// TIA Portal project "Assembler-Analog" (V15.1)

(* hardware
DEVICE "S7-1200 station_1"  S7-1200 Station
   slot 0: "Rack_0"  S7-1200 Rack  Rack  V1.0
   slot 1: "PLC_1"  CPU 1211C DC/DC/DC  6ES7 211-1AE40-0XB0  V4.2
DEVICE "HMI_1"  KTP900 Basic PN
   slot 0: "HMI_1"  KTP900 Basic PN  6AV2 123-2JB03-0AX0  15.1.0.0
   slot 1: "HMI_RT_1"  KTP900 Basic PN  6AV2 123-2JB03-0AX0  15.1.0.0
   slot 5: "HMI_1.IE_CP_1"  PROFINET Interface  15.0.1.0
      slot 1: "PROFINET Interface_1"  PROFINET Interface
         slot 1: "Port_1"  Port
*)

// ===== PLC "PLC_1"  CPU 1211C DC/DC/DC =====

VAR_GLOBAL   // PLC tag table "Default tag table"
   "Clock_Byte" AT %MB0 : Byte;
   "Clock_10Hz" AT %M0.0 : Bool;
   "Clock_5Hz" AT %M0.1 : Bool;
   "Clock_2.5Hz" AT %M0.2 : Bool;
   "Clock_2Hz" AT %M0.3 : Bool;
   "Clock_1.25Hz" AT %M0.4 : Bool;
   "Clock_1Hz" AT %M0.5 : Bool;
   "Clock_0.625Hz" AT %M0.6 : Bool;
   "Clock_0.5Hz" AT %M0.7 : Bool;
END_VAR

VAR_GLOBAL   // PLC tag table "IO_tags"
   "item_detected" AT %I0.0 : Bool;
   "lid_at_place" AT %I0.1 : Bool;
   "base_at_place" AT %I0.2 : Bool;
   "part_leaving" AT %I0.3 : Bool;
   "start" AT %I0.4 : Bool;
   "reset" AT %I0.5 : Bool;
   "stop" AT %I0.6 : Bool;
   "esd" AT %I0.7 : Bool;
   "auto" AT %I1.0 : Bool;
   "running" AT %I1.1 : Bool;
   "lids_conveyor_1" AT %Q0.0 : Bool;
   "stop_blade_1" AT %Q0.1 : Bool;
   "lids_conveyor_2" AT %Q0.2 : Bool;
   "base_conveyor_1" AT %Q0.3 : Bool;
   "stop_blade_2" AT %Q0.4 : Bool;
   "base_conveyor_2" AT %Q0.5 : Bool;
   "grab" AT %Q0.6 : Bool;
   "start_light" AT %Q0.7 : Bool;
   "reset_light" AT %Q1.0 : Bool;
   "stop_light" AT %Q1.1 : Bool;
   "x" AT %ID30 : Real;
   "z" AT %ID34 : Real;
   "set_x" AT %QD30 : Real;
   "set_z" AT %QD34 : Real;
   "counter" AT %QD38 : DInt;
END_VAR

DATA_BLOCK "Auxiliare"   // DB1
{ S7_Optimized_Access := 'TRUE' }
VERSION : 0.1
   VAR
      aux_1 : Bool;
      aux_2 : Bool;
      aux_3 : Bool;
      aux_4 : Bool;
      aux_5 : Bool;
      btn_reset_counter : Bool;
   END_VAR
BEGIN
END_DATA_BLOCK

DATA_BLOCK "Alarme"   // DB2
{ S7_Optimized_Access := 'TRUE' }
VERSION : 0.1
   VAR
      gather : Word;
      "array" : Array[0..15] of Bool;
   END_VAR
BEGIN
END_DATA_BLOCK

// folder: System blocks/Program resources

DATA_BLOCK "timer_reset_counter"   // DB3
{ S7_Optimized_Access := 'TRUE' }
AUTHOR : Simatic
FAMILY : IEC
NAME : IEC_TMR
VERSION : 1.0
// stored: InstanceOfName IEC_TIMER
"IEC_TIMER"
BEGIN
END_DATA_BLOCK

// folder: (top level)

FUNCTION "Analog_Assembler" : Void   // FC1, LAD
{ S7_Optimized_Access := 'TRUE' }
VERSION : 0.1
   VAR_TEMP   // added for the SCL form of the ladder/FBD networks
      _w1 : Bool;
      _w2 : Bool;
   END_VAR
BEGIN

REGION Network 1
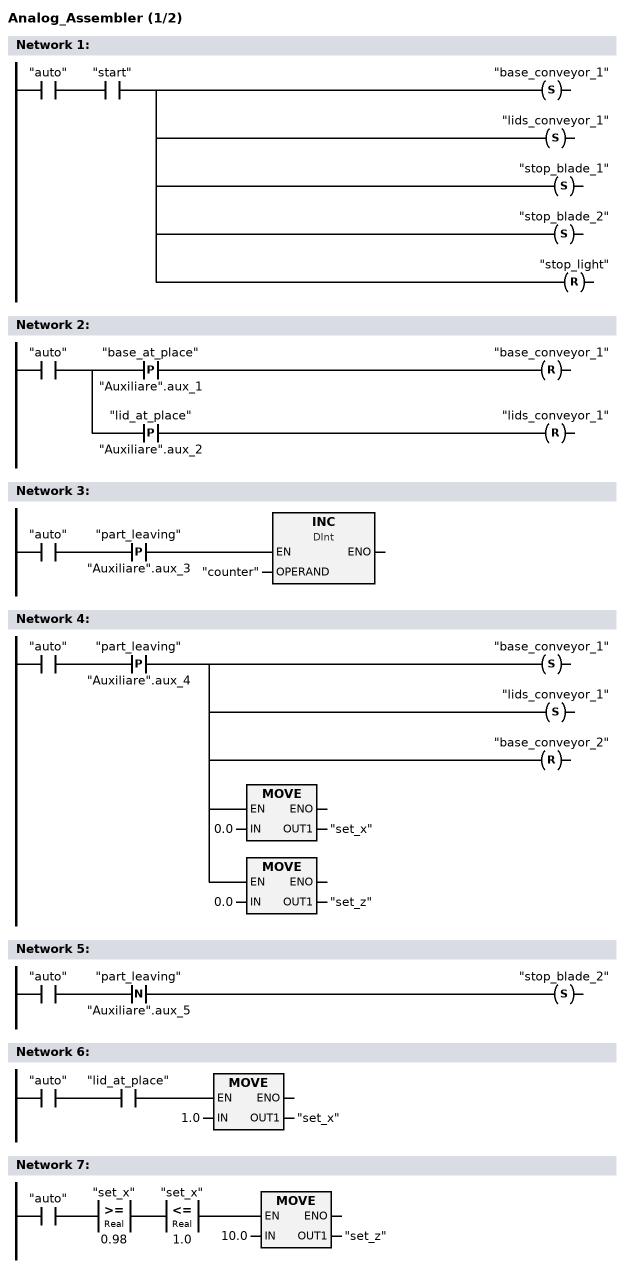
   RUNG wire#powerrail
      Contact( "auto" )
      Contact( "start" )
      wire#w1
      S_Coil( "base_conveyor_1" )
   END_RUNG
   RUNG wire#w1
      S_Coil( "lids_conveyor_1" )
   END_RUNG
   RUNG wire#w1
      S_Coil( "stop_blade_1" )
   END_RUNG
   RUNG wire#w1
      S_Coil( "stop_blade_2" )
   END_RUNG
   RUNG wire#w1
      R_Coil( "stop_light" )
   END_RUNG
   // the same network as SCL:
   IF "auto" AND "start" THEN
       "base_conveyor_1" := TRUE;
       "lids_conveyor_1" := TRUE;
       "stop_blade_1" := TRUE;
       "stop_blade_2" := TRUE;
       "stop_light" := FALSE;
   END_IF;
END_REGION

REGION Network 2
   RUNG wire#powerrail
      Contact( "auto" )
      wire#w1
      P_Contact(operand := "base_at_place", bit := "Auxiliare".aux_1)
      R_Coil( "base_conveyor_1" )
   END_RUNG
   RUNG wire#w1
      P_Contact(operand := "lid_at_place", bit := "Auxiliare".aux_2)
      R_Coil( "lids_conveyor_1" )
   END_RUNG
   // the same network as SCL:
   #_w1 := "auto" AND "base_at_place" AND NOT "Auxiliare".aux_1;   // rising edge of "base_at_place"
   "Auxiliare".aux_1 := "base_at_place";
   IF #_w1 THEN "base_conveyor_1" := FALSE; END_IF;
   #_w2 := "auto" AND "lid_at_place" AND NOT "Auxiliare".aux_2;   // rising edge of "lid_at_place"
   "Auxiliare".aux_2 := "lid_at_place";
   IF #_w2 THEN "lids_conveyor_1" := FALSE; END_IF;
END_REGION

REGION Network 3
   RUNG wire#powerrail
      Contact( "auto" )
      P_Contact(operand := "part_leaving", bit := "Auxiliare".aux_3)
      { S7_Templates := "DestType := DInt" } Inc( "counter" )
   END_RUNG
   // the same network as SCL:
   #_w1 := "auto" AND "part_leaving" AND NOT "Auxiliare".aux_3;   // rising edge of "part_leaving"
   "Auxiliare".aux_3 := "part_leaving";
   IF #_w1 THEN "counter" := "counter" + 1; END_IF;
END_REGION

REGION Network 4
   RUNG wire#powerrail
      Contact( "auto" )
      P_Contact(operand := "part_leaving", bit := "Auxiliare".aux_4)
      wire#w1
      S_Coil( "base_conveyor_1" )
   END_RUNG
   RUNG wire#w1
      S_Coil( "lids_conveyor_1" )
   END_RUNG
   RUNG wire#w1
      R_Coil( "base_conveyor_2" )
   END_RUNG
   RUNG wire#w1
      Move(in := 0.0, out1 => "set_x")
   END_RUNG
   RUNG wire#w1
      Move(in := 0.0, out1 => "set_z")
   END_RUNG
   // the same network as SCL:
   #_w1 := "auto" AND "part_leaving" AND NOT "Auxiliare".aux_4;   // rising edge of "part_leaving"
   "Auxiliare".aux_4 := "part_leaving";
   IF #_w1 THEN
       "base_conveyor_1" := TRUE;
       "lids_conveyor_1" := TRUE;
       "base_conveyor_2" := FALSE;
       "set_x" := 0.0;
       "set_z" := 0.0;
   END_IF;
END_REGION

REGION Network 5
   RUNG wire#powerrail
      Contact( "auto" )
      N_Contact(operand := "part_leaving", bit := "Auxiliare".aux_5)
      S_Coil( "stop_blade_2" )
   END_RUNG
   // the same network as SCL:
   #_w1 := "auto" AND NOT "part_leaving" AND "Auxiliare".aux_5;   // falling edge of "part_leaving"
   "Auxiliare".aux_5 := "part_leaving";
   IF #_w1 THEN "stop_blade_2" := TRUE; END_IF;
END_REGION

REGION Network 6
   RUNG wire#powerrail
      Contact( "auto" )
      Contact( "lid_at_place" )
      Move(in := 1.0, out1 => "set_x")
   END_RUNG
   // the same network as SCL:
   IF "auto" AND "lid_at_place" THEN "set_x" := 1.0; END_IF;
END_REGION

REGION Network 7
   RUNG wire#powerrail
      Contact( "auto" )
      { S7_Templates := "SrcType := Real" } GE_Contact(in1 := "set_x", in2 := 0.98)
      { S7_Templates := "SrcType := Real" } LE_Contact(in1 := "set_x", in2 := 1.0)
      Move(in := 10.0, out1 => "set_z")
   END_RUNG
   // the same network as SCL:
   IF "auto" AND ("set_x" >= 0.98) AND ("set_x" <= 1.0) THEN "set_z" := 10.0; END_IF;
END_REGION

REGION Network 8
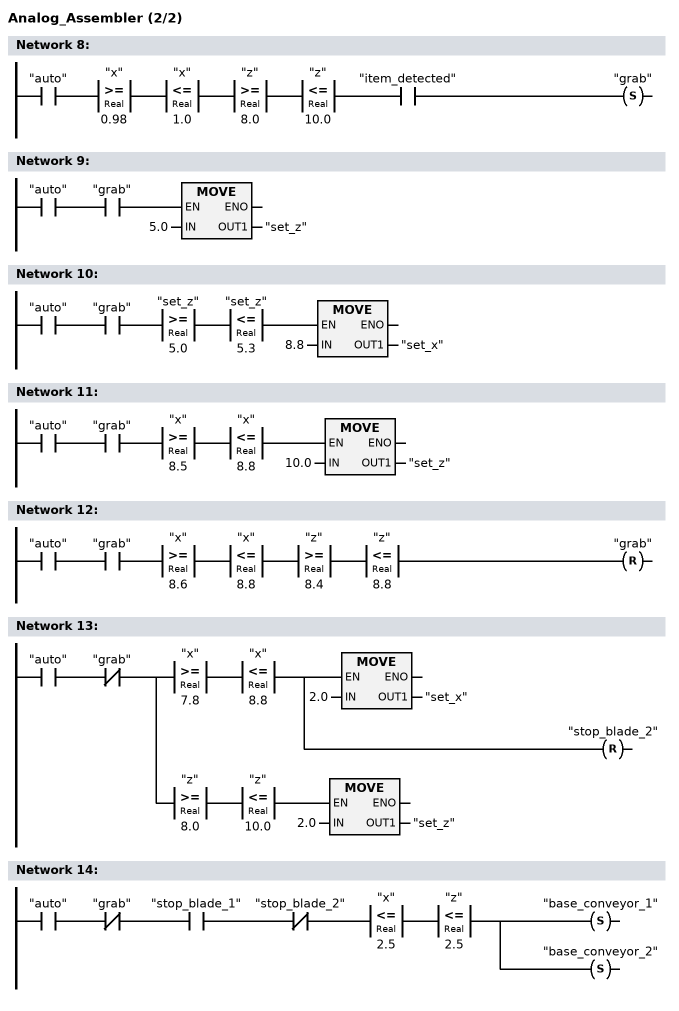
   RUNG wire#powerrail
      Contact( "auto" )
      { S7_Templates := "SrcType := Real" } GE_Contact(in1 := "x", in2 := 0.98)
      { S7_Templates := "SrcType := Real" } LE_Contact(in1 := "x", in2 := 1.0)
      { S7_Templates := "SrcType := Real" } GE_Contact(in1 := "z", in2 := 8.0)
      { S7_Templates := "SrcType := Real" } LE_Contact(in1 := "z", in2 := 10.0)
      Contact( "item_detected" )
      S_Coil( "grab" )
   END_RUNG
   // the same network as SCL:
   IF "auto" AND ("x" >= 0.98) AND ("x" <= 1.0) AND ("z" >= 8.0) AND ("z" <= 10.0) AND "item_detected" THEN
       "grab" := TRUE;
   END_IF;
END_REGION

REGION Network 9
   RUNG wire#powerrail
      Contact( "auto" )
      Contact( "grab" )
      Move(in := 5.0, out1 => "set_z")
   END_RUNG
   // the same network as SCL:
   IF "auto" AND "grab" THEN "set_z" := 5.0; END_IF;
END_REGION

REGION Network 10
   RUNG wire#powerrail
      Contact( "auto" )
      Contact( "grab" )
      { S7_Templates := "SrcType := Real" } GE_Contact(in1 := "set_z", in2 := 5.0)
      { S7_Templates := "SrcType := Real" } LE_Contact(in1 := "set_z", in2 := 5.3)
      Move(in := 8.8, out1 => "set_x")
   END_RUNG
   // the same network as SCL:
   IF "auto" AND "grab" AND ("set_z" >= 5.0) AND ("set_z" <= 5.3) THEN "set_x" := 8.8; END_IF;
END_REGION

REGION Network 11
   RUNG wire#powerrail
      Contact( "auto" )
      Contact( "grab" )
      { S7_Templates := "SrcType := Real" } GE_Contact(in1 := "x", in2 := 8.5)
      { S7_Templates := "SrcType := Real" } LE_Contact(in1 := "x", in2 := 8.8)
      Move(in := 10.0, out1 => "set_z")
   END_RUNG
   // the same network as SCL:
   IF "auto" AND "grab" AND ("x" >= 8.5) AND ("x" <= 8.8) THEN "set_z" := 10.0; END_IF;
END_REGION

REGION Network 12
   RUNG wire#powerrail
      Contact( "auto" )
      Contact( "grab" )
      { S7_Templates := "SrcType := Real" } GE_Contact(in1 := "x", in2 := 8.6)
      { S7_Templates := "SrcType := Real" } LE_Contact(in1 := "x", in2 := 8.8)
      { S7_Templates := "SrcType := Real" } GE_Contact(in1 := "z", in2 := 8.4)
      { S7_Templates := "SrcType := Real" } LE_Contact(in1 := "z", in2 := 8.8)
      R_Coil( "grab" )
   END_RUNG
   // the same network as SCL:
   IF "auto" AND "grab" AND ("x" >= 8.6) AND ("x" <= 8.8) AND ("z" >= 8.4) AND ("z" <= 8.8) THEN
       "grab" := FALSE;
   END_IF;
END_REGION

REGION Network 13
   RUNG wire#powerrail
      Contact( "auto" )
      I_Contact( "grab" )
      wire#w1
      { S7_Templates := "SrcType := Real" } GE_Contact(in1 := "x", in2 := 7.8)
      { S7_Templates := "SrcType := Real" } LE_Contact(in1 := "x", in2 := 8.8)
      wire#w2
      Move(in := 2.0, out1 => "set_x")
   END_RUNG
   RUNG wire#w2
      R_Coil( "stop_blade_2" )
   END_RUNG
   RUNG wire#w1
      { S7_Templates := "SrcType := Real" } GE_Contact(in1 := "z", in2 := 8.0)
      { S7_Templates := "SrcType := Real" } LE_Contact(in1 := "z", in2 := 10.0)
      Move(in := 2.0, out1 => "set_z")
   END_RUNG
   // the same network as SCL:
   #_w1 := "auto" AND NOT "grab";
   IF #_w1 AND ("x" >= 7.8) AND ("x" <= 8.8) THEN
       "set_x" := 2.0;
       "stop_blade_2" := FALSE;
   END_IF;
   IF #_w1 AND ("z" >= 8.0) AND ("z" <= 10.0) THEN "set_z" := 2.0; END_IF;
END_REGION

REGION Network 14
   RUNG wire#powerrail
      Contact( "auto" )
      I_Contact( "grab" )
      Contact( "stop_blade_1" )
      I_Contact( "stop_blade_2" )
      { S7_Templates := "SrcType := Real" } LE_Contact(in1 := "x", in2 := 2.5)
      { S7_Templates := "SrcType := Real" } LE_Contact(in1 := "z", in2 := 2.5)
      wire#w1
      S_Coil( "base_conveyor_1" )
   END_RUNG
   RUNG wire#w1
      S_Coil( "base_conveyor_2" )
   END_RUNG
   // the same network as SCL:
   IF "auto" AND NOT "grab" AND "stop_blade_1" AND NOT "stop_blade_2" AND ("x" <= 2.5) AND ("z" <= 2.5) THEN
       "base_conveyor_1" := TRUE;
       "base_conveyor_2" := TRUE;
   END_IF;
END_REGION
END_FUNCTION

FUNCTION "MHJ-PLC-Lab-Function-S71200" : Void   // FC9000, SCL
{ S7_Optimized_Access := 'TRUE' }
VERSION : 0.1
   VAR_TEMP
      rdTimeReturn : Int;
      outputTime : DTL;
      SyncVal : Byte;
      forVal : Int;
      forVal_2 : Int;
      Value : Byte;
   END_VAR
   VAR CONSTANT
      CompVal : Byte := 16#34;
      Value_01 : Byte := 16#11;
      Value_01_DW : DWord := 16#A165_D992;
      Value_02_DW : DWord := 16#58BE_4401;
   END_VAR
BEGIN

   #Value:=PEEK(area := 16#82,
        dbNumber := 0,
        byteOffset := 511);
   #Value := #Value + 1;

   POKE(area := 16#82,
        dbNumber := 0,
        byteOffset := 511,
        value := #Value);

   POKE(area:=16#81,
        dbNumber:=0,
        byteOffset:=1016,
        value:=#Value_01_DW);
   POKE(area := 16#81,
        dbNumber := 0,
        byteOffset := 1020,
        value := #Value_02_DW);

   POKE(area := 16#81,
        dbNumber := 0,
        byteOffset := 511,
        value := B#16#00);

   FOR #forVal := 0 TO 120 DO
       FOR #forVal_2:=0 TO 10 DO
           #rdTimeReturn:=RD_SYS_T(#outputTime);
           #rdTimeReturn := WR_SYS_T(#outputTime);
           #rdTimeReturn := RD_SYS_T(#outputTime);
           #rdTimeReturn := WR_SYS_T(#outputTime);
       END_FOR;
       #SyncVal:= PEEK(area := 16#81,
                      dbNumber := 0,
                      byteOffset := 511);
       IF #SyncVal = #CompVal THEN
          GOTO M_1;
       END_IF;
   END_FOR;
   RETURN;

   M_1:
   POKE(area := 16#81,
        dbNumber := 0,
        byteOffset := 511,
        value := B#16#0);
END_FUNCTION

ORGANIZATION_BLOCK "Main"   // OB1, LAD, ProgramCycle
TITLE = "Main Program Sweep (Cycle)"
{ S7_Optimized_Access := 'TRUE' }
VERSION : 0.1
   VAR_INPUT
      Initial_Call : Bool;   // Initial call of this OB
      Remanence : Bool;   // =True, if remanent data are available
   END_VAR
BEGIN

REGION Network 1: fct de conectare la factory io
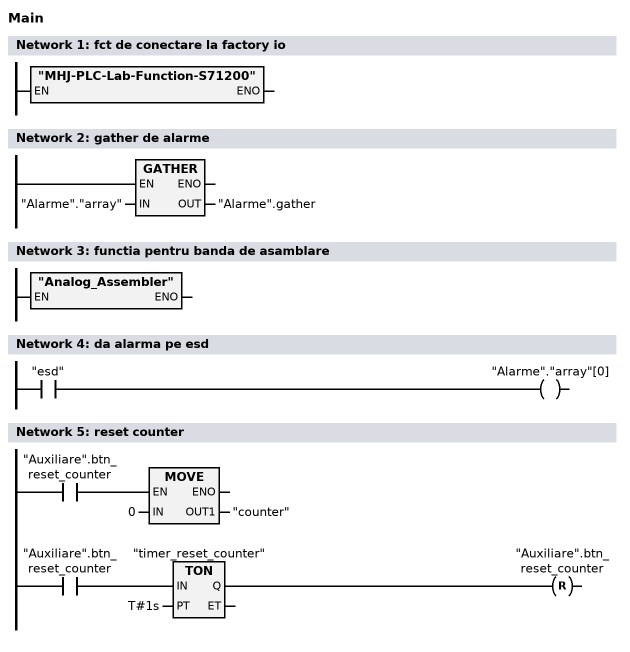
   RUNG wire#powerrail
      "MHJ-PLC-Lab-Function-S71200"()
   END_RUNG
   // the same network as SCL:
   "MHJ-PLC-Lab-Function-S71200"();
END_REGION

REGION Network 2: gather de alarme
   GATHER(IN := "Alarme"."array", OUT => "Alarme".gather);
END_REGION

REGION Network 3: functia pentru banda de asamblare
   RUNG wire#powerrail
      "Analog_Assembler"()
   END_RUNG
   // the same network as SCL:
   "Analog_Assembler"();
END_REGION

REGION Network 4: da alarma pe esd
   RUNG wire#powerrail
      Contact( "esd" )
      Coil( "Alarme"."array"[0] )
   END_RUNG
   // the same network as SCL:
   "Alarme"."array"[0] := "esd";
END_REGION

REGION Network 5: reset counter
   IF "Auxiliare".btn_reset_counter THEN "counter" := 0; END_IF;
   "timer_reset_counter".TON(IN := "Auxiliare".btn_reset_counter, PT := T#1s);
   IF "timer_reset_counter".Q THEN "Auxiliare".btn_reset_counter := FALSE; END_IF;
END_REGION
END_ORGANIZATION_BLOCK

(* ===== HMI "HMI_RT_1" =====
system functions are stored by id; their names below are inferred from use
connection "HMI_Connection_1": ETHERNET, SMART_S7_1200_OMS

HMI tags "Default tag table"
   "counter" : DInt = PLC counter AT %QD38, 1 s
   "Auxiliare_btn_reset_counter" : Bool = PLC Auxiliare.btn_reset_counter, 1 s
   "Alarme_gather" : Word = PLC Alarme.gather, 1 s

discrete alarms
   1: 'ESD', class Errors, trigger "Alarme_gather" bit 0

Template "Template_1" 800x480
   Button "Exit" at 722,440 size 55x39; TextOff 'Exit'; PictureOff "ExitRuntime_KTP900_Basic_PN_TR"; PictureOn "ExitRuntime_KTP900_Basic_PN_TR"
      on Release: StopRuntime(0)
   Button "Template_Button" at 622,440 size 55x39; TextOff 'Text'
   Button "Template_Button_1" at 522,440 size 55x39; TextOff 'Text'
   Button "Template_Button_2" at 422,440 size 55x39; TextOff 'Text'
   Button "Template_Button_3" at 322,440 size 55x39; TextOff 'Text'
   Button "Template_Button_4" at 222,440 size 55x39; TextOff 'Text'
   Button "Template_Button_5" at 122,440 size 55x39; TextOff 'Text'
   Button "Template_Button_6" at 22,440 size 55x39; TextOff 'Text'

screen "Main" 800x480, template "Template_1"
   IOField "I/O field_1" at 308,126 size 200x71; FormatPattern 99999
      ProcessValue <- "counter"
   TextField "Text field_1" at 355,90 size 105x34; Text 'Counter'
   Button "Button_1" at 365,209 size 96x32; TextOff 'Reset'
      on Click: SetBit("Auxiliare_btn_reset_counter")
*)